// TIA Portal V16 export
// export: Created 2020-12-17T10:22:04.9411875Z, ExportSetting WithReadOnly, DisplayName Totally Integrated Automation Portal, DisplayVersion V16 Update 2, DisplayName TIA Portal Version Control Interface, DisplayVersion V16 Update 2, DisplayName TIA Portal Openness, DisplayVersion V16 Update 2, DisplayName STEP 7 Professional, DisplayVersion V16 Update 2, DisplayName STEP 7 Safety, DisplayVersion V16, DisplayName WinCC Advanced / Unified PC, DisplayVersion V16 Update 2
FUNCTION "Block_S1" : Void   // FC3, SCL
{ S7_Optimized_Access := 'TRUE' }
// stored: CodeModifiedDate 2020-12-17T10:18:16.964766Z, CompileDate 2020-12-17T10:18:16.964766Z, CreationDate 2020-12-17T10:17:02.6275941Z, InterfaceModifiedDate 2020-12-17T10:17:32.4776481Z, IsConsistent true, LibraryConformanceStatus The object is library-conformant., ModifiedDate 2020-12-17T10:18:16.964766Z, ParameterModified 2020-12-17T10:17:32.4776481Z, SetENOAutomatically false, StructureModified 2020-12-17T10:17:32.4776481Z
   VAR_INPUT
      iEnable : Bool;
      iStart : Int;
   END_VAR
   VAR_IN_OUT
      ioCount : Int;
   END_VAR
BEGIN
   IF #iEnable THEN
       #ioCount := #ioCount + 1;
   ELSE
       #ioCount := #iStart;
   END_IF;
END_FUNCTION
